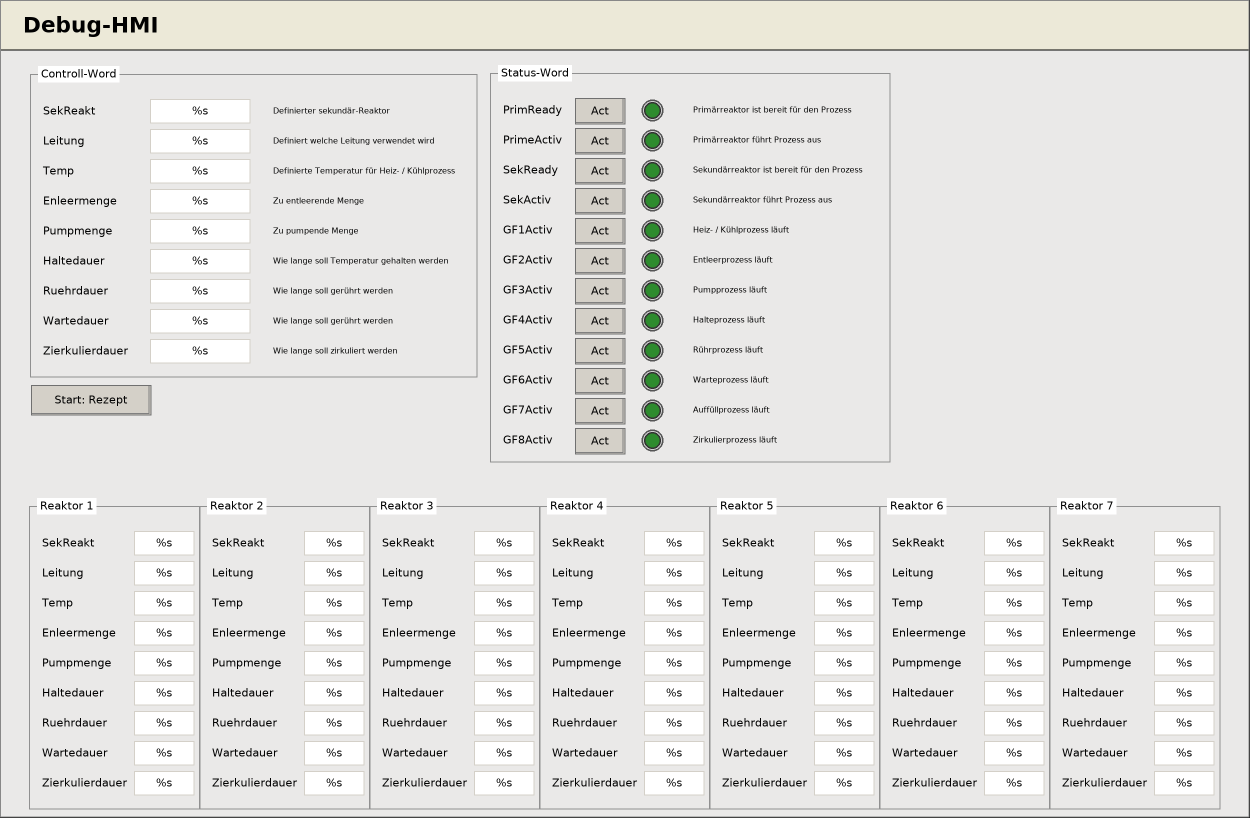
VISUALIZATION Debug_Visu  // 1250x818
    Rectangle (0,0 1250x818)
    Rectangle (0,0 1250x50)
    Label (20,0 1230x50), "Debug-HMI"
    GroupBox (30,66 447x311), "Controll-Word"
        Label (10,30 150x30), "SekReakt"
        Label (10,60 150x30), "Leitung"
        Label (10,90 150x30), "Temp"
        Label (10,120 150x30), "Enleermenge"
        Label (10,150 150x30), "Pumpmenge"
        Label (10,180 150x30), "Haltedauer"
        Label (10,210 150x30), "Ruehrdauer"
        Label (10,240 150x30), "Wartedauer"
        Label (10,270 150x30), "Zierkulierdauer"
        Textfield (120,33 100x24), "%s", text variable: GVL.Param_CW.SekReakt
            OnMouseClick: write GVL.Param_CW.SekReakt via Edit
        Textfield (120,63 100x24), "%s", text variable: GVL.Param_CW.Leitung
            OnMouseClick: write GVL.Param_CW.Leitung via Edit
        Textfield (120,93 100x24), "%s", text variable: GVL.Param_CW.Temp
            OnMouseClick: write GVL.Param_CW.Temp via Edit
        Textfield (120,123 100x24), "%s", text variable: GVL.Param_CW.Enlteermenge
            OnMouseClick: write GVL.Param_CW.Enlteermenge via Edit
        Textfield (120,153 100x24), "%s", text variable: GVL.Param_CW.Pumpmenge
            OnMouseClick: write GVL.Param_CW.Pumpmenge via Edit
        Textfield (120,183 100x24), "%s", text variable: GVL.Param_CW.Haltedauer
            OnMouseClick: write GVL.Param_CW.Haltedauer via Edit
        Textfield (120,213 100x24), "%s", text variable: GVL.Param_CW.Ruehrdauer
            OnMouseClick: write GVL.Param_CW.Ruehrdauer via Edit
        Textfield (120,243 100x24), "%s", text variable: GVL.Param_CW.Wartedauer
            OnMouseClick: write GVL.Param_CW.Wartedauer via Edit
        Textfield (120,273 100x24), "%s", text variable: GVL.Param_CW.Zirkulierdauer
            OnMouseClick: write GVL.Param_CW.Zirkulierdauer via Edit
        Label (240,30 300x30), "Definierter sekundär-Reaktor"
        Label (240,60 300x30), "Definiert welche Leitung verwendet wird"
        Label (240,90 300x30), "Definierte Temperatur für Heiz- / Kühlprozess"
        Label (240,120 300x30), "Zu entleerende Menge"
        Label (240,150 300x30), "Zu pumpende Menge"
        Label (240,180 300x30), "Wie lange soll Temperatur gehalten werden"
        Label (240,210 300x30), "Wie lange soll gerührt werden"
        Label (240,240 300x30), "Wie lange soll gerührt werden"
        Label (240,270 300x30), "Wie lange soll zirkuliert werden"
    GroupBox (490,65 400x397), "Status-Word"
        Label (10,30 150x30), "PrimReady"
        Label (10,60 150x30), "PrimeActiv"
        Label (10,90 150x30), "SekReady"
        Label (10,120 150x30), "SekActiv"
        Label (10,150 150x30), "GF1Activ"
        Label (10,180 150x30), "GF2Activ"
        Label (10,210 150x30), "GF3Activ"
        Label (10,240 150x30), "GF4Activ"
        Label (10,270 150x30), "GF5Activ"
        Label (200,30 300x30), "Primärreaktor ist bereit für den Prozess"
        Label (200,60 300x30), "Primärreaktor führt Prozess aus"
        Label (200,90 300x30), "Sekundärreaktor ist bereit für den Prozess"
        Label (200,120 300x30), "Sekundärreaktor führt Prozess aus"
        Label (200,150 300x30), "Heiz- / Kühlprozess läuft"
        Label (200,180 300x30), "Entleerprozess läuft"
        Label (200,210 300x30), "Pumpprozess läuft"
        Label (200,240 300x30), "Halteprozess läuft"
        Label (200,270 300x30), "Rührprozess läuft"
        Label (10,300 150x30), "GF6Activ"
        Label (10,330 150x30), "GF7Activ"
        Label (10,360 150x30), "GF8Activ"
        Button (85,33 50x26), "Act"
            toggle GVL.Debug_SW.PrimReady
        Lamp1 (150,33 25x25), variable: GVL.Debug_SW.PrimReady, style: Lamp-Lamp1-Green
        Button (85,63 50x26), "Act"
            toggle GVL.Debug_SW.PrimActiv
        Button (85,93 50x26), "Act"
            toggle GVL.Debug_SW.SekReady
        Button (85,123 50x26), "Act"
            toggle GVL.Debug_SW.SekActiv
        Button (85,153 50x26), "Act"
            toggle GVL.Debug_SW.GF1Activ
        Button (85,183 50x26), "Act"
            toggle GVL.Debug_SW.GF2Activ
        Button (85,213 50x26), "Act"
            toggle GVL.Debug_SW.GF3Activ
        Button (85,243 50x26), "Act"
            toggle GVL.Debug_SW.GF4Activ
        Button (85,273 50x26), "Act"
            toggle GVL.Debug_SW.GF5Activ
        Button (85,303 50x26), "Act"
            toggle GVL.Debug_SW.GF6Activ
        Button (85,333 50x26), "Act"
            toggle GVL.Debug_SW.GF7Activ
        Button (85,363 50x26), "Act"
            toggle GVL.Debug_SW.GF8Activ
        Lamp1 (150,63 25x25), variable: GVL.Debug_SW.PrimActiv, style: Lamp-Lamp1-Green
        Lamp1 (150,93 25x25), variable: GVL.Debug_SW.SekReady, style: Lamp-Lamp1-Green
        Lamp1 (150,123 25x25), variable: GVL.Debug_SW.SekActiv, style: Lamp-Lamp1-Green
        Lamp1 (150,153 25x25), variable: GVL.Debug_SW.GF1Activ, style: Lamp-Lamp1-Green
        Lamp1 (150,183 25x25), variable: GVL.Debug_SW.GF2Activ, style: Lamp-Lamp1-Green
        Lamp1 (150,213 25x25), variable: GVL.Debug_SW.GF3Activ, style: Lamp-Lamp1-Green
        Lamp1 (150,243 25x25), variable: GVL.Debug_SW.GF4Activ, style: Lamp-Lamp1-Green
        Lamp1 (150,273 25x25), variable: GVL.Debug_SW.GF5Activ, style: Lamp-Lamp1-Green
        Lamp1 (150,303 25x25), variable: GVL.Debug_SW.GF6Activ, style: Lamp-Lamp1-Green
        Lamp1 (150,333 25x25), variable: GVL.Debug_SW.GF7Activ, style: Lamp-Lamp1-Green
        Lamp1 (150,363 25x25), variable: GVL.Debug_SW.GF8Activ, style: Lamp-Lamp1-Green
    Label (690,365 300x30), "Warteprozess läuft"
    Label (690,395 300x30), "Auffüllprozess läuft"
    Label (690,425 300x30), "Zirkulierprozess läuft"
    GroupBox (29,498 171x311), "Reaktor 1"
        Label (10,30 150x30), "SekReakt"
        Label (10,60 150x30), "Leitung"
        Label (10,90 150x30), "Temp"
        Label (10,120 150x30), "Enleermenge"
        Label (10,150 150x30), "Pumpmenge"
        Label (10,180 150x30), "Haltedauer"
        Label (10,210 150x30), "Ruehrdauer"
        Label (10,240 150x30), "Wartedauer"
        Label (10,270 150x30), "Zierkulierdauer"
        Textfield (105,33 60x24), "%s", text variable: GVL.RZCW_R1.SekReakt, input disabled if: TRUE
        Textfield (105,63 60x24), "%s", text variable: GVL.RZCW_R1.Leitung, input disabled if: TRUE
        Textfield (105,93 60x24), "%s", text variable: GVL.RZCW_R1.Temp, input disabled if: TRUE
        Textfield (105,123 60x24), "%s", text variable: GVL.RZCW_R1.Enlteermenge, input disabled if: TRUE
        Textfield (105,153 60x24), "%s", text variable: GVL.RZCW_R1.Pumpmenge, input disabled if: TRUE
        Textfield (105,183 60x24), "%s", text variable: GVL.RZCW_R1.Haltedauer, input disabled if: TRUE
        Textfield (105,213 60x24), "%s", text variable: GVL.RZCW_R1.Ruehrdauer, input disabled if: TRUE
        Textfield (105,243 60x24), "%s", text variable: GVL.RZCW_R1.Wartedauer, input disabled if: TRUE
        Textfield (105,273 60x24), "%s", text variable: GVL.RZCW_R1.Zirkulierdauer, input disabled if: TRUE
    Button (31,385 120x30), "Start: Rezept"
        OnMouseClick: toggle GVL.Start
    GroupBox (199,498 171x311), "Reaktor 2"
        Label (10,30 150x30), "SekReakt"
        Label (10,60 150x30), "Leitung"
        Label (10,90 150x30), "Temp"
        Label (10,120 150x30), "Enleermenge"
        Label (10,150 150x30), "Pumpmenge"
        Label (10,180 150x30), "Haltedauer"
        Label (10,210 150x30), "Ruehrdauer"
        Label (10,240 150x30), "Wartedauer"
        Label (10,270 150x30), "Zierkulierdauer"
        Textfield (105,33 60x24), "%s", text variable: GVL.RZCW_R2.SekReakt, input disabled if: TRUE
        Textfield (105,63 60x24), "%s", text variable: GVL.RZCW_R2.Leitung, input disabled if: TRUE
        Textfield (105,93 60x24), "%s", text variable: GVL.RZCW_R2.Temp, input disabled if: TRUE
        Textfield (105,123 60x24), "%s", text variable: GVL.RZCW_R2.Enlteermenge, input disabled if: TRUE
        Textfield (105,153 60x24), "%s", text variable: GVL.RZCW_R2.Pumpmenge, input disabled if: TRUE
        Textfield (105,183 60x24), "%s", text variable: GVL.RZCW_R2.Haltedauer, input disabled if: TRUE
        Textfield (105,213 60x24), "%s", text variable: GVL.RZCW_R2.Ruehrdauer, input disabled if: TRUE
        Textfield (105,243 60x24), "%s", text variable: GVL.RZCW_R2.Wartedauer, input disabled if: TRUE
        Textfield (105,273 60x24), "%s", text variable: GVL.RZCW_R2.Zirkulierdauer, input disabled if: TRUE
    GroupBox (369,498 171x311), "Reaktor 3"
        Label (10,30 150x30), "SekReakt"
        Label (10,60 150x30), "Leitung"
        Label (10,90 150x30), "Temp"
        Label (10,120 150x30), "Enleermenge"
        Label (10,150 150x30), "Pumpmenge"
        Label (10,180 150x30), "Haltedauer"
        Label (10,210 150x30), "Ruehrdauer"
        Label (10,240 150x30), "Wartedauer"
        Label (10,270 150x30), "Zierkulierdauer"
        Textfield (105,33 60x24), "%s", text variable: GVL.RZCW_R3.SekReakt, input disabled if: TRUE
        Textfield (105,63 60x24), "%s", text variable: GVL.RZCW_R3.Leitung, input disabled if: TRUE
        Textfield (105,93 60x24), "%s", text variable: GVL.RZCW_R3.Temp, input disabled if: TRUE
        Textfield (105,123 60x24), "%s", text variable: GVL.RZCW_R3.Enlteermenge, input disabled if: TRUE
        Textfield (105,153 60x24), "%s", text variable: GVL.RZCW_R3.Pumpmenge, input disabled if: TRUE
        Textfield (105,183 60x24), "%s", text variable: GVL.RZCW_R3.Haltedauer, input disabled if: TRUE
        Textfield (105,213 60x24), "%s", text variable: GVL.RZCW_R3.Ruehrdauer, input disabled if: TRUE
        Textfield (105,243 60x24), "%s", text variable: GVL.RZCW_R3.Wartedauer, input disabled if: TRUE
        Textfield (105,273 60x24), "%s", text variable: GVL.RZCW_R3.Zirkulierdauer, input disabled if: TRUE
    GroupBox (539,498 171x311), "Reaktor 4"
        Label (10,30 150x30), "SekReakt"
        Label (10,60 150x30), "Leitung"
        Label (10,90 150x30), "Temp"
        Label (10,120 150x30), "Enleermenge"
        Label (10,150 150x30), "Pumpmenge"
        Label (10,180 150x30), "Haltedauer"
        Label (10,210 150x30), "Ruehrdauer"
        Label (10,240 150x30), "Wartedauer"
        Label (10,270 150x30), "Zierkulierdauer"
        Textfield (105,33 60x24), "%s", text variable: GVL.RZCW_R4.SekReakt, input disabled if: TRUE
        Textfield (105,63 60x24), "%s", text variable: GVL.RZCW_R4.Leitung, input disabled if: TRUE
        Textfield (105,93 60x24), "%s", text variable: GVL.RZCW_R4.Temp, input disabled if: TRUE
        Textfield (105,123 60x24), "%s", text variable: GVL.RZCW_R4.Enlteermenge, input disabled if: TRUE
        Textfield (105,153 60x24), "%s", text variable: GVL.RZCW_R4.Pumpmenge, input disabled if: TRUE
        Textfield (105,183 60x24), "%s", text variable: GVL.RZCW_R4.Haltedauer, input disabled if: TRUE
        Textfield (105,213 60x24), "%s", text variable: GVL.RZCW_R4.Ruehrdauer, input disabled if: TRUE
        Textfield (105,243 60x24), "%s", text variable: GVL.RZCW_R4.Wartedauer, input disabled if: TRUE
        Textfield (105,273 60x24), "%s", text variable: GVL.RZCW_R4.Zirkulierdauer, input disabled if: TRUE
    GroupBox (709,498 171x311), "Reaktor 5"
        Label (10,30 150x30), "SekReakt"
        Label (10,60 150x30), "Leitung"
        Label (10,90 150x30), "Temp"
        Label (10,120 150x30), "Enleermenge"
        Label (10,150 150x30), "Pumpmenge"
        Label (10,180 150x30), "Haltedauer"
        Label (10,210 150x30), "Ruehrdauer"
        Label (10,240 150x30), "Wartedauer"
        Label (10,270 150x30), "Zierkulierdauer"
        Textfield (105,33 60x24), "%s", text variable: GVL.RZCW_R5.SekReakt, input disabled if: TRUE
        Textfield (105,63 60x24), "%s", text variable: GVL.RZCW_R5.Leitung, input disabled if: TRUE
        Textfield (105,93 60x24), "%s", text variable: GVL.RZCW_R5.Temp, input disabled if: TRUE
        Textfield (105,123 60x24), "%s", text variable: GVL.RZCW_R5.Enlteermenge, input disabled if: TRUE
        Textfield (105,153 60x24), "%s", text variable: GVL.RZCW_R5.Pumpmenge, input disabled if: TRUE
        Textfield (105,183 60x24), "%s", text variable: GVL.RZCW_R5.Haltedauer, input disabled if: TRUE
        Textfield (105,213 60x24), "%s", text variable: GVL.RZCW_R5.Ruehrdauer, input disabled if: TRUE
        Textfield (105,243 60x24), "%s", text variable: GVL.RZCW_R5.Wartedauer, input disabled if: TRUE
        Textfield (105,273 60x24), "%s", text variable: GVL.RZCW_R5.Zirkulierdauer, input disabled if: TRUE
    GroupBox (879,498 171x311), "Reaktor 6"
        Label (10,30 150x30), "SekReakt"
        Label (10,60 150x30), "Leitung"
        Label (10,90 150x30), "Temp"
        Label (10,120 150x30), "Enleermenge"
        Label (10,150 150x30), "Pumpmenge"
        Label (10,180 150x30), "Haltedauer"
        Label (10,210 150x30), "Ruehrdauer"
        Label (10,240 150x30), "Wartedauer"
        Label (10,270 150x30), "Zierkulierdauer"
        Textfield (105,33 60x24), "%s", text variable: GVL.RZCW_R6.SekReakt, input disabled if: TRUE
        Textfield (105,63 60x24), "%s", text variable: GVL.RZCW_R6.Leitung, input disabled if: TRUE
        Textfield (105,93 60x24), "%s", text variable: GVL.RZCW_R6.Temp, input disabled if: TRUE
        Textfield (105,123 60x24), "%s", text variable: GVL.RZCW_R6.Enlteermenge, input disabled if: TRUE
        Textfield (105,153 60x24), "%s", text variable: GVL.RZCW_R6.Pumpmenge, input disabled if: TRUE
        Textfield (105,183 60x24), "%s", text variable: GVL.RZCW_R6.Haltedauer, input disabled if: TRUE
        Textfield (105,213 60x24), "%s", text variable: GVL.RZCW_R6.Ruehrdauer, input disabled if: TRUE
        Textfield (105,243 60x24), "%s", text variable: GVL.RZCW_R6.Wartedauer, input disabled if: TRUE
        Textfield (105,273 60x24), "%s", text variable: GVL.RZCW_R6.Zirkulierdauer, input disabled if: TRUE
    GroupBox (1049,498 171x311), "Reaktor 7"
        Label (10,30 150x30), "SekReakt"
        Label (10,60 150x30), "Leitung"
        Label (10,90 150x30), "Temp"
        Label (10,120 150x30), "Enleermenge"
        Label (10,150 150x30), "Pumpmenge"
        Label (10,180 150x30), "Haltedauer"
        Label (10,210 150x30), "Ruehrdauer"
        Label (10,240 150x30), "Wartedauer"
        Label (10,270 150x30), "Zierkulierdauer"
        Textfield (105,33 60x24), "%s", text variable: GVL.RZCW_R7.SekReakt, input disabled if: TRUE
        Textfield (105,63 60x24), "%s", text variable: GVL.RZCW_R7.Leitung, input disabled if: TRUE
        Textfield (105,93 60x24), "%s", text variable: GVL.RZCW_R7.Temp, input disabled if: TRUE
        Textfield (105,123 60x24), "%s", text variable: GVL.RZCW_R7.Enlteermenge, input disabled if: TRUE
        Textfield (105,153 60x24), "%s", text variable: GVL.RZCW_R7.Pumpmenge, input disabled if: TRUE
        Textfield (105,183 60x24), "%s", text variable: GVL.RZCW_R7.Haltedauer, input disabled if: TRUE
        Textfield (105,213 60x24), "%s", text variable: GVL.RZCW_R7.Ruehrdauer, input disabled if: TRUE
        Textfield (105,243 60x24), "%s", text variable: GVL.RZCW_R7.Wartedauer, input disabled if: TRUE
        Textfield (105,273 60x24), "%s", text variable: GVL.RZCW_R7.Zirkulierdauer, input disabled if: TRUE
END_VISUALIZATION

(* stored: Version 1.1.0.1, ProductVersion 3.1.4024.12
   Visu Debug_Visu: Id {7a986ea6-c035-4ae4-8912-39bf6be96f2f} *)
